// TIA Portal V19 export
FUNCTION "OutputHandler1" : Void   // FC51, STL
{ S7_Optimized_Access := 'TRUE' }
AUTHOR : FLA
FAMILY : UHT
VERSION : 1.0
// Programmer Init: 8953-FLA
// 
// Change Log:
// 
// Date        Change                          Updated by
// ------------------------------------------------------
// 19.04.99    1. Edition                      FLA
// stored: AutoNumber false
BEGIN

NETWORK
TITLE = 
// Item control
// Y0101, NC, Product inlet valve, with 2 feed-back
      CALL  "Item_Control"
      ( "type"      := 3,  // 0=NO-FB, 1=SET-FB, 2=RES-FB, 3=S/R-FB
        maxTime     := 8,  // Max feed-back MAX_TIME
        itemInfo    := "ItemInfoScada".Items[1],  //Y0101
        itemTimer   := "ItemTimerwork".Y0101,
        itemStatus  := "ItemStatus".Y0101,
        itemCommand := "ItemCommand".Y0101,
        resetInput  := "Y0101R",  // Input for de-energised feed-back
        setInput    := "Y0101S",  // Input for energised feed-back
        output      := "Y0101"  // Output
      );

NETWORK
TITLE = 
// Item control
// Y0103, NC, Cip / steam inlet valve, with 2 feed-back
      CALL  "Item_Control"
      ( "type"      := 3,  // 0=NO-FB, 1=SET-FB, 2=RES-FB, 3=S/R-FB
        maxTime     := 8,  // Max feed-back MAX_TIME
        itemInfo    := "ItemInfoScada".Items[2],  //Y0103
        itemTimer   := "ItemTimerwork".Y0103,
        itemStatus  := "ItemStatus".Y0103,
        itemCommand := "ItemCommand".Y0103,
        resetInput  := "Y0103R",  // Input for de-energised feed-back
        setInput    := "Y0103S",  // Input for energised feed-back
        output      := "Y0103"  // Output
      );


NETWORK
TITLE = 
// Item control
// Y0104, NC, Cip / steam inlet valve, with 2 feed-back
      CALL  "Item_Control"
      ( "type"      := 3,  // 0=NO-FB, 1=SET-FB, 2=RES-FB, 3=S/R-FB
        maxTime     := 8,  // Max feed-back MAX_TIME
        itemInfo    := "ItemInfoScada".Items[3],  //Y0104
        itemTimer   := "ItemTimerwork".Y0104,
        itemStatus  := "ItemStatus".Y0104,
        itemCommand := "ItemCommand".Y0104,
        resetInput  := "Y0104R",  // Input for de-energised feed-back
        setInput    := "Y0104S",  // Input for energised feed-back
        output      := "Y0104"  // Output
      );

NETWORK
TITLE = 
// Item control
// Y0109, NO, Cooling water to jacket valve, with 2 feed-back
      CALL  "Item_Control"
      ( "type"      := 3,  // 0=NO-FB, 1=SET-FB, 2=RES-FB, 3=S/R-FB
        maxTime     := 8,  // Max feed-back MAX_TIME
        itemInfo    := "ItemInfoScada".Items[4],  //Y0109
        itemTimer   := "ItemTimerwork".Y0109,
        itemStatus  := "ItemStatus".Y0109,
        itemCommand := "ItemCommand".Y0109,
        resetInput  := "Y0109R",  // Input for de-energised feed-back
        setInput    := "Y0109S",  // Input for energised feed-back
        output      := "Y0109"  // Output
      );


NETWORK
TITLE = 
// Item control
// Y0111, NO, Sterile air inlet valve, with 2 feed-back
      CALL  "Item_Control"
      ( "type"      := 3,  // 0=NO-FB, 1=SET-FB, 2=RES-FB, 3=S/R-FB
        maxTime     := 8,  // Max feed-back MAX_TIME
        itemInfo    := "ItemInfoScada".Items[5],  //Y0111
        itemTimer   := "ItemTimerwork".Y0111,
        itemStatus  := "ItemStatus".Y0111,
        itemCommand := "ItemCommand".Y0111,
        resetInput  := "Y0111R",  // Input for de-energised feed-back
        setInput    := "Y0111S",  // Input for energised feed-back
        output      := "Y0111"  // Output
      );


NETWORK
TITLE = 
// Item control
// Y0112, NC, Filling line stop valve, with 2 feed-back
      CALL  "Item_Control"
      ( "type"      := 3,  // 0=NO-FB, 1=SET-FB, 2=RES-FB, 3=S/R-FB
        maxTime     := 8,  // Max feed-back MAX_TIME
        itemInfo    := "ItemInfoScada".Items[6],  //Y0112
        itemTimer   := "ItemTimerwork".Y0112,
        itemStatus  := "ItemStatus".Y0112,
        itemCommand := "ItemCommand".Y0112,
        resetInput  := "Y0112R",  // Input for de-energised feed-back
        setInput    := "Y0112S",  // Input for energised feed-back
        output      := "Y0112"  // Output
      );


NETWORK
TITLE = 
// Item control
// Y0113, NO, Filling line steam / cip valve, with 2 feed-back
      CALL  "Item_Control"
      ( "type"      := 3,  // 0=NO-FB, 1=SET-FB, 2=RES-FB, 3=S/R-FB
        maxTime     := 8,  // Max feed-back MAX_TIME
        itemInfo    := "ItemInfoScada".Items[7],  //Y0113
        itemTimer   := "ItemTimerwork".Y0113,
        itemStatus  := "ItemStatus".Y0113,
        itemCommand := "ItemCommand".Y0113,
        resetInput  := "Y0113R",  // Input for de-energised feed-back
        setInput    := "Y0113S",  // Input for energised feed-back
        output      := "Y0113"  // Output
      );


NETWORK
TITLE = 
// Item control
// Y0114, NC, Cip return / drain valve, with 2 feed-back
      CALL  "Item_Control"
      ( "type"      := 3,  // 0=NO-FB, 1=SET-FB, 2=RES-FB, 3=S/R-FB
        maxTime     := 8,  // Max feed-back MAX_TIME
        itemInfo    := "ItemInfoScada".Items[8],  //Y0114
        itemTimer   := "ItemTimerwork".Y0114,
        itemStatus  := "ItemStatus".Y0114,
        itemCommand := "ItemCommand".Y0114,
        resetInput  := "Y0114R",  // Input for de-energised feed-back
        setInput    := "Y0114S",  // Input for energised feed-back
        output      := "Y0114"  // Output
      );


NETWORK
TITLE = 
// Item control
// Y0115, NC, Water to balance tank valve, with 2 feed-back
      CALL  "Item_Control"
      ( "type"      := 3,  // 0=NO-FB, 1=SET-FB, 2=RES-FB, 3=S/R-FB
        maxTime     := 8,  // Max feed-back MAX_TIME
        itemInfo    := "ItemInfoScada".Items[9],  //Y0115
        itemTimer   := "ItemTimerwork".Y0115,
        itemStatus  := "ItemStatus".Y0115,
        itemCommand := "ItemCommand".Y0115,
        resetInput  := "Y0115R",  // Input for de-energised feed-back
        setInput    := "Y0115S",  // Input for energised feed-back
        output      := "Y0115"  // Output
      );


NETWORK
TITLE = 
// Item control
// M0139, NO, Cip pump, with 1 feed-back
      CALL  "Item_Control"
      ( "type"      := 1,  // 0=NO-FB, 1=SET-FB, 2=RES-FB, 3=S/R-FB
        maxTime     := 10,  // Max feed-back MAX_TIME
        itemInfo    := "ItemInfoScada".Items[10],  //M0139
        itemTimer   := "ItemTimerwork".M0139,
        itemStatus  := "ItemStatus".M0139,
        itemCommand := "ItemCommand".M0139,
        resetInput  := "AFI",  // Input for de-energised feed-back
        setInput    := "M0139S",  // Input for energised feed-back
        output      := "M0139"  // Output
      );

NETWORK
TITLE = 
// Item control
// Y0116, NO, Cip return from tank/filling, with 2 feed-back
      CALL  "Item_Control"
      ( "type"      := 3,  // 0=NO-FB, 1=SET-FB, 2=RES-FB, 3=S/R-FB
        maxTime     := 8,  // Max feed-back MAX_TIME
        itemInfo    := "ItemInfoScada".Items[11],  //Y0116
        itemTimer   := "ItemTimerwork".Y0116,
        itemStatus  := "ItemStatus".Y0116,
        itemCommand := "ItemCommand".Y0116,
        resetInput  := "Y0116R",  // Input for de-energised feed-back
        setInput    := "Y0116S",  // Input for energised feed-back
        output      := "Y0116"  // Output
      );


NETWORK
TITLE = 
// Item control
// Y0108, NO, Steam / cip to valve 01.01, with 2 feed-back
      CALL  "Item_Control"
      ( "type"      := 3,  // 0=NO-FB, 1=SET-FB, 2=RES-FB, 3=S/R-FB
        maxTime     := 8,  // Max feed-back MAX_TIME
        itemInfo    := "ItemInfoScada".Items[12],  //Y0108
        itemTimer   := "ItemTimerwork".Y0108,
        itemStatus  := "ItemStatus".Y0108,
        itemCommand := "ItemCommand".Y0108,
        resetInput  := "Y0108R",  // Input for de-energised feed-back
        setInput    := "Y0108S",  // Input for energised feed-back
        output      := "Y0108"  // Output
      );


NETWORK
TITLE = 
// Item control
// Y0117, NO, Cip, with 2 feed-back
      CALL  "Item_Control"
      ( "type"      := 3,  // 0=NO-FB, 1=SET-FB, 2=RES-FB, 3=S/R-FB
        maxTime     := 8,  // Max feed-back MAX_TIME
        itemInfo    := "ItemInfoScada".Items[13],  //Y0117
        itemTimer   := "ItemTimerwork".Y0117,
        itemStatus  := "ItemStatus".Y0117,
        itemCommand := "ItemCommand".Y0117,
        resetInput  := "Y0117R",  // Input for de-energised feed-back
        setInput    := "Y0117S",  // Input for energised feed-back
        output      := "Y0117"  // Output
      );


NETWORK
TITLE = 
// Item control
// Y0118, NC, Steam valve, with 0 feed-back
      CALL  "Item_Control"
      ( "type"      := 0,  // 0=NO-FB, 1=SET-FB, 2=RES-FB, 3=S/R-FB
        maxTime     := 8,  // Max feed-back MAX_TIME
        itemInfo    := "ItemInfoScada".Items[14],  //Y0118
        itemTimer   := "ItemTimerwork".Y0118,
        itemStatus  := "ItemStatus".Y0118,
        itemCommand := "ItemCommand".Y0118,
        resetInput  := "AFI",  // Input for de-energised feed-back
        setInput    := "AFI",  // Input for energised feed-back
        output      := "Y0118"  // Output
      );

NETWORK
TITLE = 
// Item control
// Y0237, , Relay signal to uht request lye, with 0 feed-back
      CALL  "Item_Control"
      ( "type"      := 0,  // 0=NO-FB, 1=SET-FB, 2=RES-FB, 3=S/R-FB
        maxTime     := 10,  // Max feed-back MAX_TIME
        itemInfo    := "ItemInfoScada".Items[15],  //Y0237
        itemTimer   := "ItemTimerwork".Y0237,
        itemStatus  := "ItemStatus".Y0237,
        itemCommand := "ItemCommand".Y0237,
        resetInput  := "AFI",  // Input for de-energised feed-back
        setInput    := "AFI",  // Input for energised feed-back
        output      := "Y0237"  // Output
      );

NETWORK
TITLE = 
// Item control
// Y0238, , Relay signal to uht request acid, with 0 feed-back
      CALL  "Item_Control"
      ( "type"      := 0,  // 0=NO-FB, 1=SET-FB, 2=RES-FB, 3=S/R-FB
        maxTime     := 10,  // Max feed-back MAX_TIME
        itemInfo    := "ItemInfoScada".Items[16],  //Y0238
        itemTimer   := "ItemTimerwork".Y0238,
        itemStatus  := "ItemStatus".Y0238,
        itemCommand := "ItemCommand".Y0238,
        resetInput  := "AFI",  // Input for de-energised feed-back
        setInput    := "AFI",  // Input for energised feed-back
        output      := "Y0238"  // Output
      );


NETWORK
TITLE = 
// Item control
// Y0119, NO, Flush chain wash, with no feed-back ..AFL 21 Aug 07

NETWORK
TITLE = 
// Item control
// Y0124, NC, By-pass valve steam valve 01.01, with 0 feed-back
      CALL  "Item_Control"
      ( "type"      := 0,  // 0=NO-FB, 1=SET-FB, 2=RES-FB, 3=S/R-FB
        maxTime     := 10,  // Max feed-back MAX_TIME
        itemInfo    := "ItemInfoScada".Items[18],  //Y0124
        itemTimer   := "ItemTimerwork".Y0124,
        itemStatus  := "ItemStatus".Y0124,
        itemCommand := "ItemCommand".Y0124,
        resetInput  := "AFI",  // Input for de-energised feed-back
        setInput    := "AFI",  // Input for energised feed-back
        output      := "Y0124"  // Output
      );


NETWORK
TITLE = 
// Item control
// Y0135_NOT_USED, , Condensate valve agitator, with 0 feed-back
      CALL  "Item_Control"
      ( "type"      := 0,  // 0=NO-FB, 1=SET-FB, 2=RES-FB, 3=S/R-FB
        maxTime     := 10,  // Max feed-back MAX_TIME
        itemInfo    := "ItemInfoScada".Items[19],  //Y0135_NOT_USED
        itemTimer   := "ItemTimerwork".Y0135_NOT_USED,
        itemStatus  := "ItemStatus".Y0135_NOT_USED,
        itemCommand := "ItemCommand".Y0135_NOT_USED,
        resetInput  := "AFI",  // Input for de-energised feed-back
        setInput    := "AFI",  // Input for energised feed-back
        output      := "Y0135"  // Output
      );


NETWORK
TITLE = 
// Item control
// Y0136_NOT_USED, , Steam to condenstate valve, with 0 feed-back
      CALL  "Item_Control"
      ( "type"      := 0,  // 0=NO-FB, 1=SET-FB, 2=RES-FB, 3=S/R-FB
        maxTime     := 10,  // Max feed-back MAX_TIME
        itemInfo    := "ItemInfoScada".Items[20],  //Y0136_NOT_USED
        itemTimer   := "ItemTimerwork".Y0136_NOT_USED,
        itemStatus  := "ItemStatus".Y0136_NOT_USED,
        itemCommand := "ItemCommand".Y0136_NOT_USED,
        resetInput  := "AFI",  // Input for de-energised feed-back
        setInput    := "AFI",  // Input for energised feed-back
        output      := "Y0136"  // Output
      );


NETWORK
TITLE = 
// Item control
// Y0137_NOT_USED, , Water to condensater valve, with 0 feed-back
      CALL  "Item_Control"
      ( "type"      := 0,  // 0=NO-FB, 1=SET-FB, 2=RES-FB, 3=S/R-FB
        maxTime     := 10,  // Max feed-back MAX_TIME
        itemInfo    := "ItemInfoScada".Items[21],  //Y0137_NOT_USED
        itemTimer   := "ItemTimerwork".Y0137_NOT_USED,
        itemStatus  := "ItemStatus".Y0137_NOT_USED,
        itemCommand := "ItemCommand".Y0137_NOT_USED,
        resetInput  := "AFI",  // Input for de-energised feed-back
        setInput    := "AFI",  // Input for energised feed-back
        output      := "Y0137"  // Output
      );


NETWORK
TITLE = 
// Item control
// Y0143, NC, Drain valve bottom sterile filter, with 0 feed-back
      CALL  "Item_Control"
      ( "type"      := 0,  // 0=NO-FB, 1=SET-FB, 2=RES-FB, 3=S/R-FB
        maxTime     := 10,  // Max feed-back MAX_TIME
        itemInfo    := "ItemInfoScada".Items[22],  //Y0143
        itemTimer   := "ItemTimerwork".Y0143,
        itemStatus  := "ItemStatus".Y0143,
        itemCommand := "ItemCommand".Y0143,
        resetInput  := "AFI",  // Input for de-energised feed-back
        setInput    := "AFI",  // Input for energised feed-back
        output      := "Y0143"  // Output
      );


NETWORK
TITLE = 
// Item control
// Y0144_NOT_USED, NC, Drain valve cip 01.01, with 0 feed-back
      CALL  "Item_Control"
      ( "type"      := 0,  // 0=NO-FB, 1=SET-FB, 2=RES-FB, 3=S/R-FB
        maxTime     := 10,  // Max feed-back MAX_TIME
        itemInfo    := "ItemInfoScada".Items[23],  //Y0144_NOT_USED
        itemTimer   := "ItemTimerwork".Y0144_NOT_USED,
        itemStatus  := "ItemStatus".Y0144_NOT_USED,
        itemCommand := "ItemCommand".Y0144_NOT_USED,
        resetInput  := "AFI",  // Input for de-energised feed-back
        setInput    := "AFI",  // Input for energised feed-back
        output      := "Y0144"  // Output
      );


NETWORK
TITLE = 
// Item control
// Y0147, NC, Steam valve to 01.13, with 0 feed-back
      CALL  "Item_Control"
      ( "type"      := 0,  // 0=NO-FB, 1=SET-FB, 2=RES-FB, 3=S/R-FB
        maxTime     := 10,  // Max feed-back MAX_TIME
        itemInfo    := "ItemInfoScada".Items[24],  //Y0147
        itemTimer   := "ItemTimerwork".Y0147,
        itemStatus  := "ItemStatus".Y0147,
        itemCommand := "ItemCommand".Y0147,
        resetInput  := "AFI",  // Input for de-energised feed-back
        setInput    := "AFI",  // Input for energised feed-back
        output      := "Y0147"  // Output
      );


NETWORK
TITLE = 
// Item control
// Y0148, NC, Steam valve to sterilzing, with 0 feed-back
      CALL  "Item_Control"
      ( "type"      := 0,  // 0=NO-FB, 1=SET-FB, 2=RES-FB, 3=S/R-FB
        maxTime     := 10,  // Max feed-back MAX_TIME
        itemInfo    := "ItemInfoScada".Items[25],  //Y0148
        itemTimer   := "ItemTimerwork".Y0148,
        itemStatus  := "ItemStatus".Y0148,
        itemCommand := "ItemCommand".Y0148,
        resetInput  := "AFI",  // Input for de-energised feed-back
        setInput    := "AFI",  // Input for energised feed-back
        output      := "Y0148"  // Output
      );


NETWORK
TITLE = 
// Item control
// Y0158, NC, Steam valve to injector, with 0 feed-back
      CALL  "Item_Control"
      ( "type"      := 0,  // 0=NO-FB, 1=SET-FB, 2=RES-FB, 3=S/R-FB
        maxTime     := 10,  // Max feed-back MAX_TIME
        itemInfo    := "ItemInfoScada".Items[26],  //Y0158
        itemTimer   := "ItemTimerwork".Y0158,
        itemStatus  := "ItemStatus".Y0158,
        itemCommand := "ItemCommand".Y0158,
        resetInput  := "AFI",  // Input for de-energised feed-back
        setInput    := "AFI",  // Input for energised feed-back
        output      := "Y0158"  // Output
      );


NETWORK
TITLE = 
// Item control
// Y0545, NC, Steam by-pass valve reduced, with 0 feed-back
      CALL  "Item_Control"
      ( "type"      := 0,  // 0=NO-FB, 1=SET-FB, 2=RES-FB, 3=S/R-FB
        maxTime     := 10,  // Max feed-back MAX_TIME
        itemInfo    := "ItemInfoScada".Items[27],  //Y0545
        itemTimer   := "ItemTimerwork".Y0545,
        itemStatus  := "ItemStatus".Y0545,
        itemCommand := "ItemCommand".Y0545,
        resetInput  := "AFI",  // Input for de-energised feed-back
        setInput    := "AFI",  // Input for energised feed-back
        output      := "Y0545"  // Output
      );


NETWORK
TITLE = 
// Item control
// Q21_3_NotUsed, , spare, with 0 feed-back
      CALL  "Item_Control"
      ( "type"      := 0,  // 0=NO-FB, 1=SET-FB, 2=RES-FB, 3=S/R-FB
        maxTime     := 10,  // Max feed-back MAX_TIME
        itemInfo    := "ItemInfoScada".Items[28],  //PACK1
        itemTimer   := "ItemTimerwork".PACK1,
        itemStatus  := "ItemStatus".PACK1,
        itemCommand := "ItemCommand".PACK1,
        resetInput  := "AFI",  // Input for de-energised feed-back
        setInput    := "AFI",  // Input for energised feed-back
        output      := "PACK1"  // Output
      );


NETWORK
TITLE = 
// Item control
// Q21_4_NotUsed, , spare, with 0 feed-back
      CALL  "Item_Control"
      ( "type"      := 0,  // 0=NO-FB, 1=SET-FB, 2=RES-FB, 3=S/R-FB
        maxTime     := 10,  // Max feed-back MAX_TIME
        itemInfo    := "ItemInfoScada".Items[29],  //PACK2
        itemTimer   := "ItemTimerwork".PACK2,
        itemStatus  := "ItemStatus".PACK2,
        itemCommand := "ItemCommand".PACK2,
        resetInput  := "AFI",  // Input for de-energised feed-back
        setInput    := "AFI",  // Input for energised feed-back
        output      := "PACK2"  // Output
      );


NETWORK
TITLE = 
// Item control
// PACK1_2, NO, Relay signal to packing product availa., with 0 feed-back
      CALL  "Item_Control"
      ( "type"      := 0,  // 0=NO-FB, 1=SET-FB, 2=RES-FB, 3=S/R-FB
        maxTime     := 10,  // Max feed-back MAX_TIME
        itemInfo    := "ItemInfoScada".Items[30],  //PACK3
        itemTimer   := "ItemTimerwork".PACK3,
        itemStatus  := "ItemStatus".PACK3,
        itemCommand := "ItemCommand".PACK3,
        resetInput  := "AFI",  // Input for de-energised feed-back
        setInput    := "AFI",  // Input for energised feed-back
        output      := "ProdLineBeingCleaned"  // Output
      );


NETWORK
TITLE = 
// Item control
// PACK3_4, NO, Relay signal to packing product availa., with 0 feed-back
      CALL  "Item_Control"
      ( "type"      := 0,  // 0=NO-FB, 1=SET-FB, 2=RES-FB, 3=S/R-FB
        maxTime     := 10,  // Max feed-back MAX_TIME
        itemInfo    := "ItemInfoScada".Items[31],  //PACK4
        itemTimer   := "ItemTimerwork".PACK4,
        itemStatus  := "ItemStatus".PACK4,
        itemCommand := "ItemCommand".PACK4,
        resetInput  := "AFI",  // Input for de-energised feed-back
        setInput    := "AFI",  // Input for energised feed-back
        output      := "Time Stop CIP"  // Output
      );


NETWORK
TITLE = 
// Item control
// AlarmLamp, NO, Internal alarmlamp, with 0 feed-back
      CALL  "Item_Control"
      ( "type"      := 0,  // 0=NO-FB, 1=SET-FB, 2=RES-FB, 3=S/R-FB
        maxTime     := 10,  // Max feed-back MAX_TIME
        itemInfo    := "ItemInfoScada".Items[32],  //AlarmLamp
        itemTimer   := "ItemTimerwork".AlarmLamp,
        itemStatus  := "ItemStatus".AlarmLamp,
        itemCommand := "ItemCommand".AlarmLamp,
        resetInput  := "AFI",  // Input for de-energised feed-back
        setInput    := "AFI",  // Input for energised feed-back
        output      := "CIP Release"  // Output
      );

END_FUNCTION
